PROGRAM MAIN
VAR
END_VAR

END_PROGRAM

(* stored: Version 1.1.0.1, ProductVersion 3.1.4024.14
   POU MAIN: Id {928fbce8-0202-4ead-8676-e2345e284aa3}, SpecialFunc None *)
